// TIA Portal V15.1 export
// export: Created 2024-05-17T05:38:41.2840198Z, ExportSetting WithDefaults, DisplayName Totally Integrated Automation Portal, DisplayVersion V15.1 Update 5, DisplayName TIA Portal Openness, DisplayVersion V15.1 Update 5, DisplayName SINAMICS Startdrive Advanced, DisplayVersion V15.1, DisplayName G130, G150, S120, S150, SINAMICS MV, S210, DisplayVersion V15.1, DisplayName G110M, G120, G120C, G120D, G120P, DisplayVersion V15.1, DisplayName STEP 7 Professional, DisplayVersion V15.1 Update 5, DisplayName STEP 7 Safety, DisplayVersion V15.1, DisplayName WinCC Professional, DisplayVersion V15.1 Update 5, DisplayName SIMATIC Visualization Architect, DisplayVersion V15.1
FUNCTION "LGBMovUnit2Pos2W1S4Det-MoviFitFCPN-Config" : Void   // FC6654, FBD
TITLE = LMovUnit2Pos1S-C-Config / LGBMovUnit2Pos2W1S4Det-MoviFitFCPN-Config
{ S7_Optimized_Access := 'FALSE' }
AUTHOR : VCC
FAMILY : Control
NAME : Bit2Word
VERSION : 1.0
// =============================================================================
// Move Configuration 
// =============================================================================
// stored: AutoNumber false, IsIECCheckEnabled false, SetENOAutomatically False, UDAEnableTagReadback false
   VAR_INPUT
      C_ForceManual : Bool;   // Force Manual Enabled
      C_AlarmResetUsed : Bool;   // Set position / If true, the Alarms will be stored untill reseted
      C_EnableMemBegin : Bool;   // Reset position / Enable memory Begin (Command Request is memorised until pos reached)
      C_EnIntlkAlm : Bool;   // Active / Enable interlock Alarm
      C_KeepPosition : Bool;   // Invisible / If true, the last position shall be kept ON and checked
      C_EnAlmDet : Bool;   // Object out of use / Enable Alarm
      C_EnAlmOvertime : Bool;   // Object out of use / Enable Alarm
      C_MotorProtectionNc : Bool;   // Motor Protection NC contact
      C_MotorProtectionUsed : Bool;   // Motor Protection used
      C_ReleaseBrakeUsed : Bool;   // Release brake used
      C_MotionStopUsed : Bool;   // Motion Stop used
      C_AlarmHighSeverity : Bool;   // Interlock alarm for Set direction / Alarm severity
      C_InitDirection : Bool;   // Initial direction
      C_SetReset : Bool;   // Set Reset
      C_HoldPosSetDelayTime : Bool;   // Hold Position Set Delay Time
      C_HoldPosResetDelayTime : Bool;   // Hold Position Reset Delay Time
      C_ManualClampCmdSet : Bool;   // Manual Clamp Command Set
      C_ManualClampCmdReset : Bool;   // Manual Clamp Command Reset
      C_SafetySensorUsed : Bool;   // Configuration / Safety Sensor Used
      C_PosSetDelayTime : DInt;   // Set position delay timer / Set Position Delay Timer
      C_PosResDelayTime : DInt;   // Reset position delay timer / Reset Position Delay Timer
      C_RunTimeMaxSetWarn : DInt;   // Maximum Time (x1ms) that the function may run (create overtime) / Maximum Time (x1ms) that the function may run (create Overtime)
      C_RunTimeMaxSetAlarm : DInt;   // Maximum Time (x1ms) that the function may run (create overtime) / Maximum Time (x1ms) that the function may run (create Overtime)
      C_RunTimeMaxResWarn : DInt;   // Maximum Time (x1ms) that the function may run (create overtime) / Maximum Time (x1ms) that the function may run (create Overtime)
      C_RunTimeMaxResAlarm : DInt;   // Maximum Time (x1ms) that the function may run (create overtime) / Maximum Time (x1ms) that the function may run (create Overtime)
      C_TimeAlmFilt : DInt;   // Timer before any actuator alarm will be active (welding..) / Timer before any actuator Alarm will be active (welding..)
      C_Ramp : Time;   // Ramp
      C_ReferenceMotorCurrent : Real;   // Reference value for current
      C_ReferenceDriveCurrent : Real;   // Reference value for drive
      C_HWSubInput : HW_SUBMODULE;   // I/O
      C_HWSubOutput : HW_SUBMODULE;   // I/O
      C_HWSubInputStatus : HW_SUBMODULE;   // I/O
      C_EnableAlarmHW : Bool;   // Enable Alarm hardware (e.g. safetyswitch, motorprotector, detections)
   END_VAR
   VAR_IN_OUT
      IO_Config : "MovUnit2Pos-MoviFitFCPNConfig";   // Output Word
   END_VAR
BEGIN

REGION Network 1: **** 1 - Inputs **** Configuration / **** 1 - Inputs **** Move Bit Config
   // Configuration
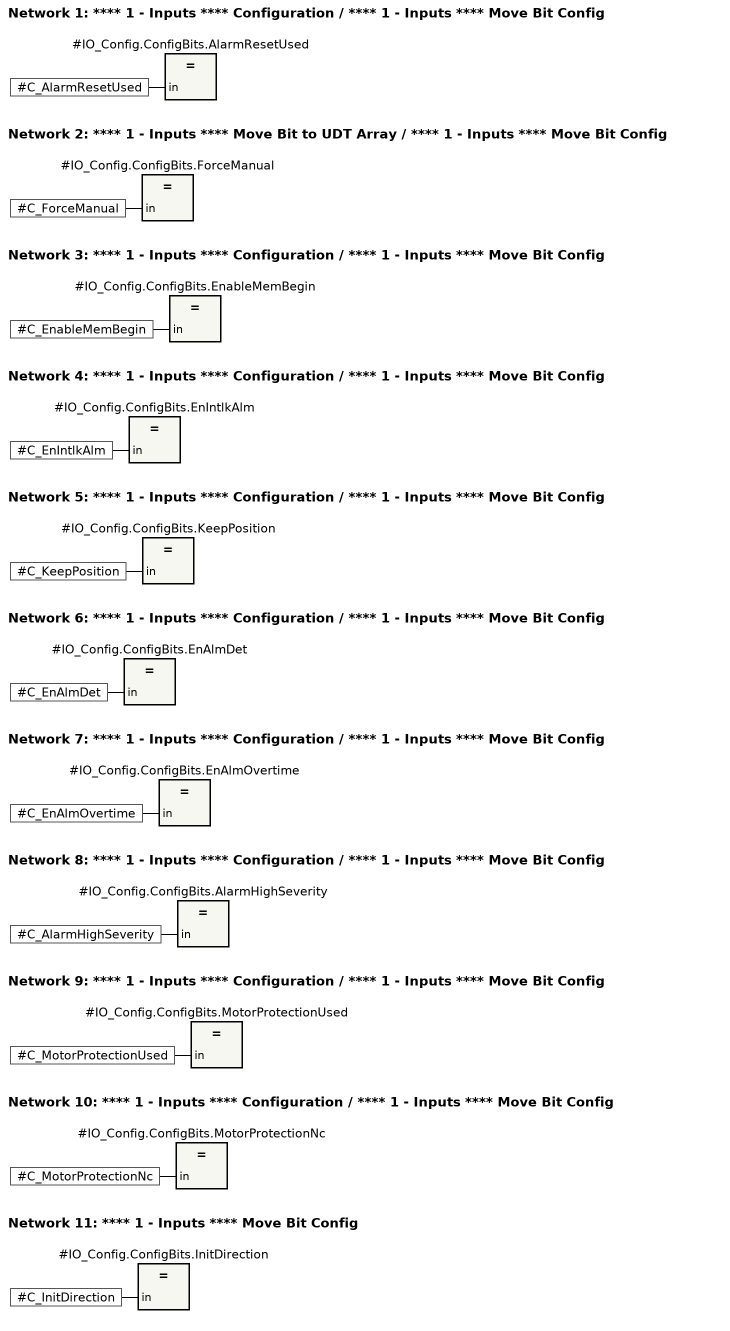
   #IO_Config.ConfigBits.AlarmResetUsed := #C_AlarmResetUsed;
END_REGION

REGION Network 2: **** 1 - Inputs **** Move Bit to UDT Array / **** 1 - Inputs **** Move Bit Config
   // Move Bit  to UDT Array
   #IO_Config.ConfigBits.ForceManual := #C_ForceManual;
END_REGION

REGION Network 3: **** 1 - Inputs **** Configuration / **** 1 - Inputs **** Move Bit Config
   // Configuration
   #IO_Config.ConfigBits.EnableMemBegin := #C_EnableMemBegin;
END_REGION

REGION Network 4: **** 1 - Inputs **** Configuration / **** 1 - Inputs **** Move Bit Config
   // Configuration
   #IO_Config.ConfigBits.EnIntlkAlm := #C_EnIntlkAlm;
END_REGION

REGION Network 5: **** 1 - Inputs **** Configuration / **** 1 - Inputs **** Move Bit Config
   // Configuration
   #IO_Config.ConfigBits.KeepPosition := #C_KeepPosition;
END_REGION

REGION Network 6: **** 1 - Inputs **** Configuration / **** 1 - Inputs **** Move Bit Config
   // Configuration
   #IO_Config.ConfigBits.EnAlmDet := #C_EnAlmDet;
END_REGION

REGION Network 7: **** 1 - Inputs **** Configuration / **** 1 - Inputs **** Move Bit Config
   // Configuration
   #IO_Config.ConfigBits.EnAlmOvertime := #C_EnAlmOvertime;
END_REGION

REGION Network 8: **** 1 - Inputs **** Configuration / **** 1 - Inputs **** Move Bit Config
   // Configuration
   #IO_Config.ConfigBits.AlarmHighSeverity := #C_AlarmHighSeverity;
END_REGION

REGION Network 9: **** 1 - Inputs **** Configuration / **** 1 - Inputs **** Move Bit Config
   // Configuration
   #IO_Config.ConfigBits.MotorProtectionUsed := #C_MotorProtectionUsed;
END_REGION

REGION Network 10: **** 1 - Inputs **** Configuration / **** 1 - Inputs **** Move Bit Config
   // Configuration
   #IO_Config.ConfigBits.MotorProtectionNc := #C_MotorProtectionNc;
END_REGION

REGION Network 11: **** 1 - Inputs **** Move Bit Config
   // Move Bit Config
   #IO_Config.ConfigBits.InitDirection := #C_InitDirection;
END_REGION

REGION Network 12: **** 1 - Inputs **** Configuration / **** 1 - Inputs **** Move Bit Config
   // Configuration
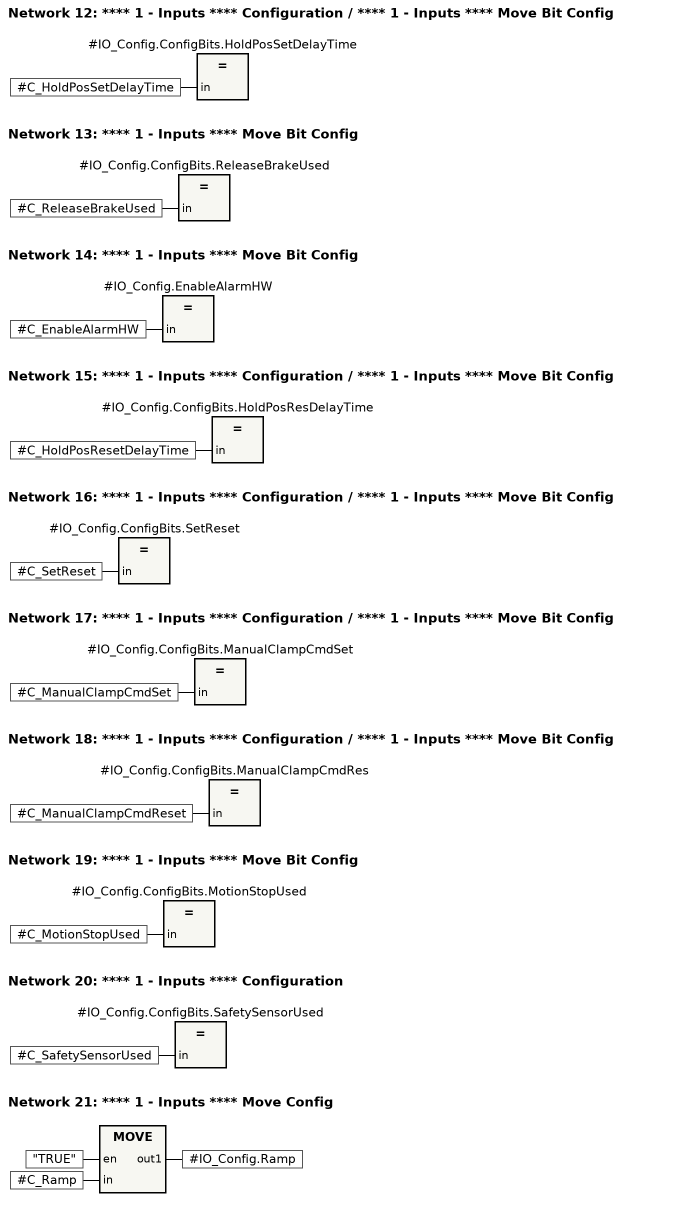
   #IO_Config.ConfigBits.HoldPosSetDelayTime := #C_HoldPosSetDelayTime;
END_REGION

REGION Network 13: **** 1 - Inputs **** Move Bit Config
   // Move Bit Config
   #IO_Config.ConfigBits.ReleaseBrakeUsed := #C_ReleaseBrakeUsed;
END_REGION

REGION Network 14: **** 1 - Inputs **** Move Bit Config
   // Move Bit Config
   #IO_Config.EnableAlarmHW := #C_EnableAlarmHW;
END_REGION

REGION Network 15: **** 1 - Inputs **** Configuration / **** 1 - Inputs **** Move Bit Config
   // Configuration
   #IO_Config.ConfigBits.HoldPosResDelayTime := #C_HoldPosResetDelayTime;
END_REGION

REGION Network 16: **** 1 - Inputs **** Configuration / **** 1 - Inputs **** Move Bit Config
   // Move bit 15Configuration
   #IO_Config.ConfigBits.SetReset := #C_SetReset;
END_REGION

REGION Network 17: **** 1 - Inputs **** Configuration / **** 1 - Inputs **** Move Bit Config
   // Configuration
   #IO_Config.ConfigBits.ManualClampCmdSet := #C_ManualClampCmdSet;
END_REGION

REGION Network 18: **** 1 - Inputs **** Configuration / **** 1 - Inputs **** Move Bit Config
   // Configuration
   #IO_Config.ConfigBits.ManualClampCmdRes := #C_ManualClampCmdReset;
END_REGION

REGION Network 19: **** 1 - Inputs **** Move Bit Config
   // Move Bit Config
   #IO_Config.ConfigBits.MotionStopUsed := #C_MotionStopUsed;
END_REGION

REGION Network 20: **** 1 - Inputs **** Configuration
   #IO_Config.ConfigBits.SafetySensorUsed := #C_SafetySensorUsed;
END_REGION

REGION Network 21: **** 1 - Inputs **** Move Config
   // Move Config
   IF "TRUE" THEN #IO_Config.Ramp := #C_Ramp; END_IF;
END_REGION

NETWORK
TITLE = **** 1 Inputs **** Move Config UDT
// Move Config
      L     #C_PosSetDelayTime;
      T     #IO_Config.PosSetDelayTime;
      L     #C_PosResDelayTime;
      T     #IO_Config.PosResDelayTime;
      L     #C_RunTimeMaxSetWarn;
      T     #IO_Config.RunTimeMaxSetWarn;
      L     #C_RunTimeMaxSetAlarm;
      T     #IO_Config.RunTimeMaxSetAlm;
      L     #C_RunTimeMaxResWarn;
      T     #IO_Config.RunTimeMaxResWarn;
      L     #C_RunTimeMaxResAlarm;
      T     #IO_Config.RunTimeMaxResAlm;
      L     #C_TimeAlmFilt;
      T     #IO_Config.TimeAlmFilt;
      L     #C_ReferenceMotorCurrent;
      T     #IO_Config.ReferenceMotorCurrent;
      L     #C_ReferenceDriveCurrent;
      T     #IO_Config.ReferenceDriveCurrent;
      L     #C_HWSubInput;
      T     #IO_Config.HWSubInput;
      L     #C_HWSubOutput;
      T     #IO_Config.HWSubOutput;
      L     #C_HWSubInputStatus;
      T     #IO_Config.HWSubInputStatus;

      L     0.0;
      T     #IO_Config.ReferenceMotorRPM;
      L     0.0;
      T     #IO_Config.RatioGearbox;
      L     0.0;
      T     #IO_Config.Diameter;
      L     0.0;
      T     #IO_Config.Acceleration;
END_FUNCTION
